{attribute 'TcGenerated'}
{attribute 'no-analysis'}
{attribute 'linkalways'}
// This function has been automatically generated from the project information.
VAR_GLOBAL CONSTANT
	{attribute 'const_non_replaced'}
	stLibVersion_ESO_LDC_Actuator_Library : ST_LibVersion := (iMajor := 1, iMinor := 0, iBuild := 0, iRevision := 2, nFlags := 0, sVersion := '1.0.0.2');
END_VAR

(* stored: Version 1.1.0.1, ProductVersion 3.1.4024.3
   GVL Global_Version: Id {5f35c67f-85a8-4dd0-8fb2-25dc162a5167} *)
